(* Ansteuerprogramm der Leitachse. Das Programm hat die Aufgabe, 
   die Leitachse in eine Bewegung konstanter Ge-schwindigkeit zu versetzen, 
   wieder anzuhalten und im Falle eines Fehlers die Achse durch einen Reset 
   wieder in einen funktionstüchtigen Zustand zu versetzen. *)

PROGRAM AbwicklerAnAus
VAR
	//stateMaster				: MoveState_t;		// Programmablauf über Zustandsvariable

	PowerAbwickler				: MC_Power;			// Schaltet Software-Freigabe der Leitachse
	PowerAbwicklerOut			: ST_McOutputs;		// 
	
	ResetAbwickler				: MC_Reset;			// Setzt Achsfehler zurück
	ResetAbwicklerOut			: ST_McOutputs;	
	
	MoveAbwickler 				: MC_MoveVelocity;	// Versetzt Leitachse in Bewegung konstanter Geschwindigkeit
	MoveAbwicklerOut			: ST_McOutputs;
	
	HaltAbwickler				: MC_Halt;			// Hält Leitachse an
	GearInAbwicklerOut: ST_McOutputs;
	HomeAbwicklerOut: ST_McOutputs;
	HaltAbwicklerOut			: ST_McOutputs;
	startAbwicklerTrig: R_TRIG;
	HaltAbwicklerTrig: R_TRIG;
	GearInAbwickler: MC_GearInDyn;
	GearOutAbwickler: MC_GearOut;
	GearOutAbwicklerOut: ST_McOutputs;
	Enable: BOOL;
	Dancer_CTL: DANCER_REF;
	Busy: BOOL;
	Error: BOOL;
	ErrorID: UDINT;
	HomeAbwickler: MC_Home;
	IntegrationCount: INT;
	PID_Methode_1: FB_BasicPID;
	GetCurrentTaskIndex: GETCURTASKINDEX;
	PIDoutput: LREAL;
	DeltaGear: LREAL := 0.005;
	GearOffset: LREAL := 1;
	PIDerrorID: UDINT;
	AbwicklerRegelungsmethode: BOOL;
	
END_VAR

//startAbwicklerTrig(clk := MaschineStart);
//HaltAbwicklerTrig(clk := Abwicklerstopp);
GlobaleVariablen.Abwickler();

CASE stateAbwickler OF
	
(* ===========================================================================================
   Zustand 1: Programm ist im Ausgangszustand und wartet auf Benutzereingabe. Alle 
   Funktionsbausteine werden initialisiert, etwaige Fehler zurückgesetzt. *)
	MOVESTATE_INIT :
		MoveAbwickler.Execute := FALSE;
		ResetAbwickler.Execute := FALSE;
		PowerAbwickler.Enable := FALSE;
		GearInAbwickler.Enable := FALSE;
		AbwicklerLaeuft := FALSE;
		IF AbwicklerStart = TRUE THEN
			stateAbwickler := MOVESTATE_ENABLE;
		END_IF

(* ===========================================================================================
   Zustand 2: Schlalten der allgemeinen Software-Freigabe, Vorschubfreigabe in positive Richtung
   durch MC_Power. Sobald Funktionsbaustein MC_Power die Betriebsbereitschaft der Achse signalisiert,
   Zustandsübergang in Forward*)
	MOVESTATE_ENABLE :
		PowerAbwickler.Enable := TRUE;
		IF PowerAbwickler.Status AND AbwicklerStart = TRUE THEN
			stateAbwickler := MOVESTATE_HOMING;
		ELSIF PowerAbwickler.Error THEN
			stateAbwickler := MOVESTATE_ERROR;
		END_IF
	
	MOVESTATE_HOMING:
		IF AbwicklerStart = TRUE AND AbwicklerStopp = FALSE THEN
			HomeAbwickler.Execute := TRUE;

			IF HomeAbwicklerOut.Done THEN
				HomeAbwickler.Execute := FALSE;
				stateAbwickler := MOVESTATE_FORWARD;
				
			ELSIF HomeAbwicklerOut.CommandAborted OR HomeAbwicklerOut.Error THEN
				stateAbwickler := MOVESTATE_ERROR;
			END_IF
		END_IF
(* ===========================================================================================
   Zustand 3: Starten des Mastern in positive Richtung mit konstanter Geschwindigkeit. 
   Zustandsübergang durch Bedienerbefehl.*)		
	MOVESTATE_FORWARD :
		IF AbwicklerStart = TRUE AND AbwicklerStopp = FALSE THEN
			GearInAbwickler.Enable := TRUE;
			
			//***********************************************************************
			//1.Methode: PID
			//***********************************************************************
			IF Master.Status.Moving AND FadenzugmotorLaeuft THEN
				PRG_PID_Abwickler();
				GlobaleVariablen.GearRatio := GearOffset + PID_Output_After_Saturation_Abwickler * DeltaGear;
			END_IF
			//***********************************************************************
			
			//***********************************************************************
			//2.Methode: Zustandsbestimmung mit integralen Ideen
			//***********************************************************************
			(*IF MasterLaeuft AND FadenzugmotorLaeuft THEN
				IF Referenzposition - Fadenzugmotor.NcToPlc.ActPos > 0 THEN
					IntegrationCount := IntegrationCount - 1;
				ELSIF Referenzposition - Fadenzugmotor.NcToPlc.ActPos < 0 THEN
					IntegrationCount := IntegrationCount + 1;
				END_IF
				
				IF IntegrationCount >= 5 THEN
					IntegrationCount := 0;
					GlobaleVariablen.GearRatio := GlobaleVariablen.GearRatio + 0.05;
				ELSIF IntegrationCount <= -5 THEN
					IntegrationCount := 0;
					GlobaleVariablen.GearRatio := GlobaleVariablen.GearRatio - 0.05;
				END_IF
			END_IF*)
			//***********************************************************************
			
			IF GlobaleVariablen.GearRatio > 1.4 THEN
				IntegrationCount := 0;
				GlobaleVariablen.GearRatio := 1.4;
			ELSIF GlobaleVariablen.GearRatio < 0.6 THEN
				IntegrationCount := 0;
				GlobaleVariablen.GearRatio := 0.6;
			END_IF
			
			IF GearInAbwicklerOut.Done THEN
				AbwicklerLaeuft := TRUE;
			END_IF
			IF GearInAbwicklerOut.CommandAborted OR GearInAbwicklerOut.Error THEN
				stateAbwickler := MOVESTATE_ERROR;
			END_IF
		ELSE
			GearInAbwickler.Enable := FALSE;
			stateAbwickler := MOVESTATE_STOPABWICKLER;
		END_IF

(* ===========================================================================================
   Zustand 4: Anhalten der Leitachse, im Anschluss Rückkehr in den Ausgangszustand. *)		
	MOVESTATE_STOPABWICKLER :
		
		IF GearOutAbwicklerOut.Done THEN
			GearOutAbwickler.Execute := FALSE;
			IF HaltAbwicklerOut.Done THEN
				HaltAbwickler.Execute := FALSE;
				AbwicklerStopp := TRUE;
				AbwicklerStart := FALSE;
				AbwicklerLaeuft := FALSE;
				stateAbwickler := MOVESTATE_INIT;
			ELSE
				HaltAbwickler.Execute := TRUE;
			END_IF
		ELSE
			GearOutAbwickler.Execute := TRUE;
		END_IF
		IF GearOutAbwicklerOut.Error OR GearOutAbwicklerOut.CommandAborted THEN
			GearOutAbwickler.Execute := FALSE;
			stateAbwickler := MOVESTATE_ERROR;
		END_IF

(* ===========================================================================================
   Zustand 5: Im Falle eines Bausteinfehlers wird überprüft, ob sich die Achse ebenfalls im    
   Fehlerzustand befindet, was einen Achsreset erfordert. Andernfalls werden Bausteinfehler 
   im Zustand Init zurückgesetzt.*)		
	MOVESTATE_ERROR :
		IF Master.Status.Error THEN
			stateAbwickler := MOVESTATE_RESET;	// Reset bei Achsfehler
		ELSE
			stateAbwickler := MOVESTATE_INIT;	// Funktionsbausteinfehler erfordert keinen Reset
		END_IF

(* ===========================================================================================
   Zustand 6:  Durchführung des Achsreset im Fehlerfall  *)		
	MOVESTATE_RESET :
		AbwicklerStart := FALSE;
		ResetAbwickler.Execute := TRUE;
		GearInAbwickler.Enable := FALSE;
		IF ResetAbwickler.Done THEN
			AbwicklerLaeuft := FALSE;
			stateAbwickler := MOVESTATE_INIT;
		ELSIF ResetAbwickler.Error THEN
			stateAbwickler := MOVESTATE_INIT; (* Falls Reset nicht gelingt, Benutzereingriff erforderlich *)
		END_IF
		
END_CASE

// Zyklusmäßige Aufrufe
ActPower();		// Aufruf des Power Funktionsbausteines
ActMove();		// Aufruf des Move-Funktionsbausteines
ActReset();		// Aufruf des Reset-Funktionsbausteines
ActHome();

ACTION ActHome:
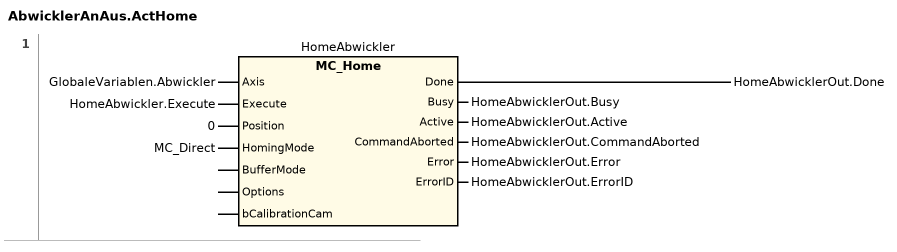
// NETWORK 1
HomeAbwickler(
    Axis := GlobaleVariablen.Abwickler,
    Execute := HomeAbwickler.Execute,
    Position := 0,
    HomingMode := MC_Direct,
    Busy => HomeAbwicklerOut.Busy,
    Active => HomeAbwicklerOut.Active,
    CommandAborted => HomeAbwicklerOut.CommandAborted,
    Error => HomeAbwicklerOut.Error,
    ErrorID => HomeAbwicklerOut.ErrorID); // MC_Home
HomeAbwicklerOut.Done := HomeAbwickler.Done;
END_ACTION

ACTION ActMove:
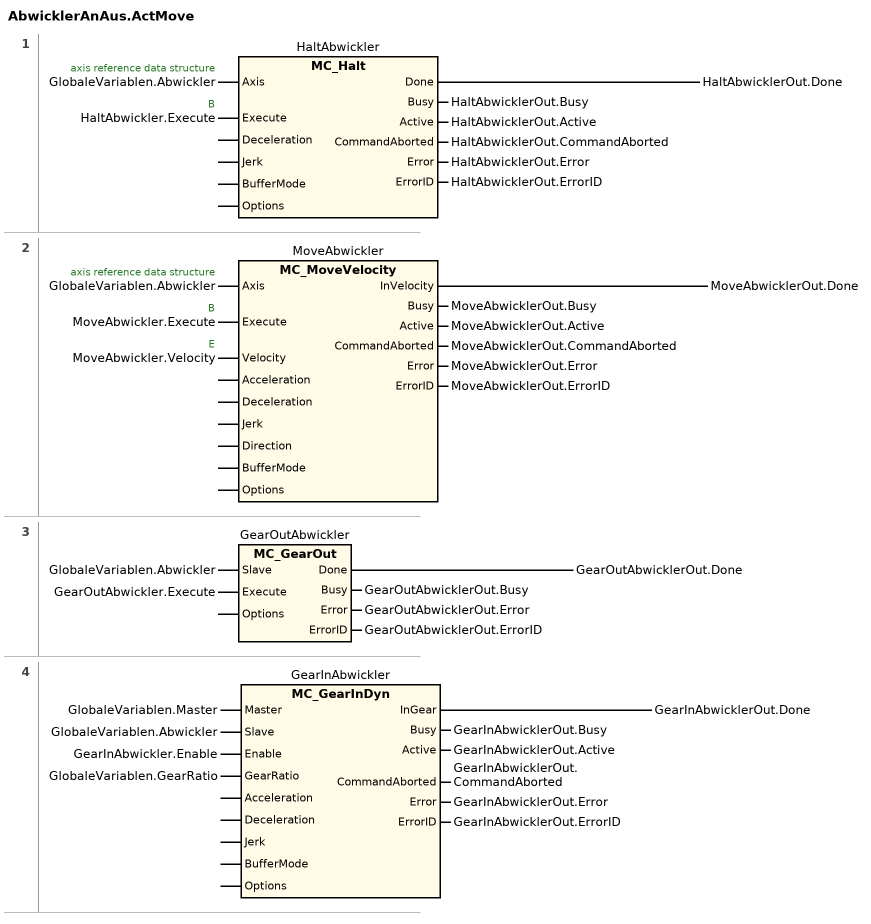
// NETWORK 1
//   GlobaleVariablen.Abwickler: axis reference data structure
//   HaltAbwickler.Execute: B
HaltAbwickler(
    Axis := GlobaleVariablen.Abwickler,
    Execute := HaltAbwickler.Execute,
    Busy => HaltAbwicklerOut.Busy,
    Active => HaltAbwicklerOut.Active,
    CommandAborted => HaltAbwicklerOut.CommandAborted,
    Error => HaltAbwicklerOut.Error,
    ErrorID => HaltAbwicklerOut.ErrorID); // MC_Halt
HaltAbwicklerOut.Done := HaltAbwickler.Done;

// NETWORK 2
//   GlobaleVariablen.Abwickler: axis reference data structure
//   MoveAbwickler.Execute: B
//   MoveAbwickler.Velocity: E
MoveAbwickler(
    Axis := GlobaleVariablen.Abwickler,
    Execute := MoveAbwickler.Execute,
    Velocity := MoveAbwickler.Velocity,
    Busy => MoveAbwicklerOut.Busy,
    Active => MoveAbwicklerOut.Active,
    CommandAborted => MoveAbwicklerOut.CommandAborted,
    Error => MoveAbwicklerOut.Error,
    ErrorID => MoveAbwicklerOut.ErrorID); // MC_MoveVelocity
MoveAbwicklerOut.Done := MoveAbwickler.InVelocity;

// NETWORK 3
GearOutAbwickler(
    Slave := GlobaleVariablen.Abwickler,
    Execute := GearOutAbwickler.Execute,
    Busy => GearOutAbwicklerOut.Busy,
    Error => GearOutAbwicklerOut.Error,
    ErrorID => GearOutAbwicklerOut.ErrorID); // MC_GearOut
GearOutAbwicklerOut.Done := GearOutAbwickler.Done;

// NETWORK 4
GearInAbwickler(
    Master := GlobaleVariablen.Master,
    Slave := GlobaleVariablen.Abwickler,
    Enable := GearInAbwickler.Enable,
    GearRatio := GlobaleVariablen.GearRatio,
    Busy => GearInAbwicklerOut.Busy,
    Active => GearInAbwicklerOut.Active,
    CommandAborted => GearInAbwicklerOut.CommandAborted,
    Error => GearInAbwicklerOut.Error,
    ErrorID => GearInAbwicklerOut.ErrorID); // MC_GearInDyn
GearInAbwicklerOut.Done := GearInAbwickler.InGear;
END_ACTION

ACTION ActPower:
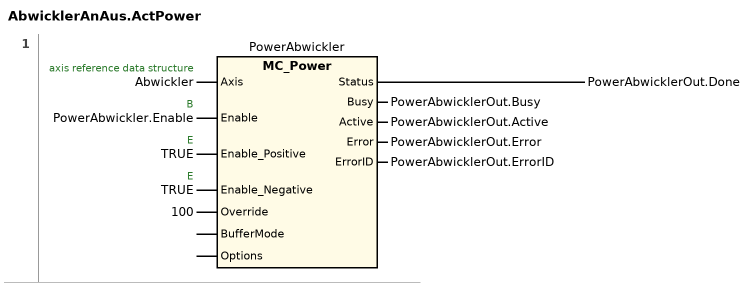
// NETWORK 1
//   Abwickler: axis reference data structure
//   PowerAbwickler.Enable: B
//   TRUE: E
PowerAbwickler(
    Axis := Abwickler,
    Enable := PowerAbwickler.Enable,
    Enable_Positive := TRUE,
    Enable_Negative := TRUE,
    Override := 100,
    Busy => PowerAbwicklerOut.Busy,
    Active => PowerAbwicklerOut.Active,
    Error => PowerAbwicklerOut.Error,
    ErrorID => PowerAbwicklerOut.ErrorID); // MC_Power
PowerAbwicklerOut.Done := PowerAbwickler.Status;
END_ACTION

ACTION ActReset:
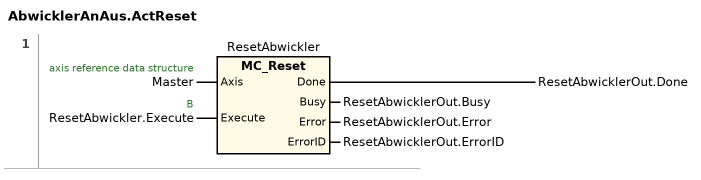
// NETWORK 1
//   Master: axis reference data structure
//   ResetAbwickler.Execute: B
ResetAbwickler(
    Axis := Master,
    Execute := ResetAbwickler.Execute,
    Busy => ResetAbwicklerOut.Busy,
    Error => ResetAbwicklerOut.Error,
    ErrorID => ResetAbwicklerOut.ErrorID); // MC_Reset
ResetAbwicklerOut.Done := ResetAbwickler.Done;
END_ACTION

END_PROGRAM

(* stored: Version 1.1.0.1, ProductVersion 3.1.4024.9
   POU AbwicklerAnAus: Id {2048ff6b-54de-4ede-a03e-a11849425f35}, SpecialFunc None
   Action ActHome: Id {69d4a677-0ea4-45a1-9512-be6d6acc0530}
   Action ActMove: Id {e2c9a395-db02-40d7-9991-207d8111ea3a}
   Action ActPower: Id {e1954218-9f22-4c53-9d48-5e065933481e}
   Action ActReset: Id {8552caf0-c0ba-43bd-897f-7d2bbc1ea57f} *)
